# EPICS substitutions: iocCollimatorControl/R15CLM.substitutions
#R15CLM_BO,EPICS->PLC,Command
file "../../db/bo_word.template"{ pattern
{	P,		R,					PORT,		OFFSET,		MASK,		ZNAM,		ONAM	}
{	SR:R15:CLM:R15CLM:,	btn_LocalOrRemote,			R15CLM_BO1_Bits,	0,		0x0001,		Low,		High	}
{	SR:R15:CLM:R15CLM:,	btn_E_STOP,				R15CLM_BO1_Bits,	0,		0x0002,		Low,		High	}
{	SR:R15:CLM:R15CLM:,	m_restartTC,				R15CLM_BO1_Bits,	0,		0x0004,		Low,		High	}
{	SR:R15:CLM:R15CLM:,	btn_Move_Axis1,				R15CLM_BO2_Bits,	0,		0x0001,		Low,		High	}
{	SR:R15:CLM:R15CLM:,	btn_JogForward_Axis1,			R15CLM_BO2_Bits,	0,		0x0002,		Low,		High	}
{	SR:R15:CLM:R15CLM:,	btn_JogBackward_Axis1,			R15CLM_BO2_Bits,	0,		0x0004,		Low,		High	}
{	SR:R15:CLM:R15CLM:,	btn_Stop_Axis1,				R15CLM_BO2_Bits,	0,		0x0008,		Low,		High	}
{	SR:R15:CLM:R15CLM:,	btn_Reset_Axis1,			R15CLM_BO2_Bits,	0,		0x0010,		Low,		High	}
{	SR:R15:CLM:R15CLM:,	btn_SetPosition_Axis1,			R15CLM_BO2_Bits,	0,		0x0020,		Low,		High	}
{	SR:R15:CLM:R15CLM:,	LVDT1_FunctionOn,			R15CLM_BO2_Bits,	0,		0x0040,		Low,		High	}
{	SR:R15:CLM:R15CLM:,	LVDT1_ManualReleaseAlarm,		R15CLM_BO2_Bits,	0,		0x0080,		Low,		High	}
{	SR:R15:CLM:R15CLM:,	btn_Move_Axis2,				R15CLM_BO3_Bits,	0,		0x0001,		Low,		High	}
{	SR:R15:CLM:R15CLM:,	btn_JogForward_Axis2,			R15CLM_BO3_Bits,	0,		0x0002,		Low,		High	}
{	SR:R15:CLM:R15CLM:,	btn_JogBackward_Axis2,			R15CLM_BO3_Bits,	0,		0x0004,		Low,		High	}
{	SR:R15:CLM:R15CLM:,	btn_Stop_Axis2,				R15CLM_BO3_Bits,	0,		0x0008,		Low,		High	}
{	SR:R15:CLM:R15CLM:,	btn_Reset_Axis2,			R15CLM_BO3_Bits,	0,		0x0010,		Low,		High	}
{	SR:R15:CLM:R15CLM:,	btn_SetPosition_Axis2,			R15CLM_BO3_Bits,	0,		0x0020,		Low,		High	}
{	SR:R15:CLM:R15CLM:,	LVDT2_FunctionOn,			R15CLM_BO3_Bits,	0,		0x0040,		Low,		High	}
{	SR:R15:CLM:R15CLM:,	LVDT2_ManualReleaseAlarm,		R15CLM_BO3_Bits,	0,		0x0080,		Low,		High	}
{	SR:R15:CLM:R15CLM:,	btn_Move_AxisAll,			R15CLM_BO4_Bits,	0,		0x0001,		Low,		High	}
{	SR:R15:CLM:R15CLM:,	btn_JogForward_AxisAll,			R15CLM_BO4_Bits,	0,		0x0002,		Low,		High	}
{	SR:R15:CLM:R15CLM:,	btn_JogBackward_AxisAll,		R15CLM_BO4_Bits,	0,		0x0004,		Low,		High	}
{	SR:R15:CLM:R15CLM:,	btn_Stop_AxisAll,			R15CLM_BO4_Bits,	0,		0x0008,		Low,		High	}
{	SR:R15:CLM:R15CLM:,	btn_Reset_AxisAll,			R15CLM_BO4_Bits,	0,		0x0010,		Low,		High	}
}
#R15CLM_AO,EPICS->PLC,Command
file "../../db/aoFloat64.template" { pattern
{	P,           	R,               			PORT,      	OFFSET,   	DATA_TYPE,    	LOPR, 	HOPR, PREC	}
{	SR:R15:CLM:R15CLM:,	targetPositionAxis1,			R15CLM_AO1_FLOAT,	0,		FLOAT32_LE,	-1e6,	1e6,	4	}
{	SR:R15:CLM:R15CLM:,	targetVelocityAxis1,			R15CLM_AO1_FLOAT,	2,		FLOAT32_LE,	-1e6,	1e6,	4	}
{	SR:R15:CLM:R15CLM:,	increaseJogPositionAxis1,		R15CLM_AO1_FLOAT,	4,		FLOAT32_LE,	-1e6,	1e6,	4	}
{	SR:R15:CLM:R15CLM:,	Axis1_minPosition,			R15CLM_AO1_FLOAT,	6,		FLOAT32_LE,	-1e6,	1e6,	4	}
{	SR:R15:CLM:R15CLM:,	Axis1_maxPosition,			R15CLM_AO1_FLOAT,	8,		FLOAT32_LE,	-1e6,	1e6,	4	}
{	SR:R15:CLM:R15CLM:,	LVDT1_Threshold,			R15CLM_AO1_FLOAT,	10,		FLOAT32_LE,	-1e6,	1e6,	4	}
{	SR:R15:CLM:R15CLM:,	PositionSetValue_Axis1,			R15CLM_AO1_FLOAT,	12,		FLOAT32_LE,	-1e6,	1e6,	4	}
{	SR:R15:CLM:R15CLM:,	targetPositionAxis2,			R15CLM_AO2_FLOAT,	0,		FLOAT32_LE,	-1e6,	1e6,	4	}
{	SR:R15:CLM:R15CLM:,	targetVelocityAxis2,			R15CLM_AO2_FLOAT,	2,		FLOAT32_LE,	-1e6,	1e6,	4	}
{	SR:R15:CLM:R15CLM:,	increaseJogPositionAxis2,		R15CLM_AO2_FLOAT,	4,		FLOAT32_LE,	-1e6,	1e6,	4	}
{	SR:R15:CLM:R15CLM:,	Axis2_minPosition,			R15CLM_AO2_FLOAT,	6,		FLOAT32_LE,	-1e6,	1e6,	4	}
{	SR:R15:CLM:R15CLM:,	Axis2_maxPosition,			R15CLM_AO2_FLOAT,	8,		FLOAT32_LE,	-1e6,	1e6,	4	}
{	SR:R15:CLM:R15CLM:,	LVDT2_Threshold,			R15CLM_AO2_FLOAT,	10,		FLOAT32_LE,	-1e6,	1e6,	4	}
{	SR:R15:CLM:R15CLM:,	PositionSetValue_Axis2,			R15CLM_AO2_FLOAT,	12,		FLOAT32_LE,	-1e6,	1e6,	4	}
}
#R15CLM_BI,PLC->EPICS,Respond
file "../../db/bi_word.template"{ pattern
{	P,		R,					PORT,		OFFSET,		MASK,		ZNAM,		ONAM,		ZSV,		OSV,		SCAN		}
{	SR:R15:CLM:R15CLM:,	E_STOP_led,				R15CLM_BI1_Bits,	0,		0x0001,		Low,		High,		NO_ALARM,	NO_ALARM,	"I/O Intr"	}
{	SR:R15:CLM:R15CLM:,	Local_led,				R15CLM_BI1_Bits,	0,		0x0002,		Low,		High,		NO_ALARM,	NO_ALARM,	"I/O Intr"	}
{	SR:R15:CLM:R15CLM:,	Remote_led,				R15CLM_BI1_Bits,	0,		0x0004,		Low,		High,		NO_ALARM,	NO_ALARM,	"I/O Intr"	}
{	SR:R15:CLM:R15CLM:,	Error_led,				R15CLM_BI1_Bits,	0,		0x0008,		Low,		High,		NO_ALARM,	NO_ALARM,	"I/O Intr"	}
{	SR:R15:CLM:R15CLM:,	Axis1_error,				R15CLM_BI2_Bits,	0,		0x0001,		Low,		High,		NO_ALARM,	NO_ALARM,	"I/O Intr"	}
{	SR:R15:CLM:R15CLM:,	Axis1_moving,				R15CLM_BI2_Bits,	0,		0x0002,		Low,		High,		NO_ALARM,	NO_ALARM,	"I/O Intr"	}
{	SR:R15:CLM:R15CLM:,	foreward_limit_axis1,			R15CLM_BI2_Bits,	0,		0x0004,		Low,		High,		NO_ALARM,	NO_ALARM,	"I/O Intr"	}
{	SR:R15:CLM:R15CLM:,	backward_limit_axis1,			R15CLM_BI2_Bits,	0,		0x0008,		Low,		High,		NO_ALARM,	NO_ALARM,	"I/O Intr"	}
{	SR:R15:CLM:R15CLM:,	Moving_done_Axis1,			R15CLM_BI2_Bits,	0,		0x0010,		Low,		High,		NO_ALARM,	NO_ALARM,	"I/O Intr"	}
{	SR:R15:CLM:R15CLM:,	PositionSetDone_Axis1,			R15CLM_BI2_Bits,	0,		0x0020,		Low,		High,		NO_ALARM,	NO_ALARM,	"I/O Intr"	}
{	SR:R15:CLM:R15CLM:,	Axis2_error,				R15CLM_BI3_Bits,	0,		0x0001,		Low,		High,		NO_ALARM,	NO_ALARM,	"I/O Intr"	}
{	SR:R15:CLM:R15CLM:,	Axis2_moving,				R15CLM_BI3_Bits,	0,		0x0002,		Low,		High,		NO_ALARM,	NO_ALARM,	"I/O Intr"	}
{	SR:R15:CLM:R15CLM:,	foreward_limit_axis2,			R15CLM_BI3_Bits,	0,		0x0004,		Low,		High,		NO_ALARM,	NO_ALARM,	"I/O Intr"	}
{	SR:R15:CLM:R15CLM:,	backward_limit_axis2,			R15CLM_BI3_Bits,	0,		0x0008,		Low,		High,		NO_ALARM,	NO_ALARM,	"I/O Intr"	}
{	SR:R15:CLM:R15CLM:,	Moving_done_Axis2,			R15CLM_BI3_Bits,	0,		0x0010,		Low,		High,		NO_ALARM,	NO_ALARM,	"I/O Intr"	}
{	SR:R15:CLM:R15CLM:,	PositionSetDone_Axis2,			R15CLM_BI3_Bits,	0,		0x0020,		Low,		High,		NO_ALARM,	NO_ALARM,	"I/O Intr"	}
}
#R15CLM_AI,PLC->EPICS,Respond
file "../../db/aiFloat64.template"{ pattern
{	P,			R,					PORT,		OFFSET,		DATA_TYPE,	LOPR,	HOPR,	PREC,	SCAN			}
{	SR:R15:CLM:R15CLM:,	Axis1_Currentvelocity,			R15CLM_AI1_FLOAT,	0,		FLOAT32_LE,	-1e6,	1e6,	4,	"I/O Intr"		}
{	SR:R15:CLM:R15CLM:,	Axis1_CurrentPosition,			R15CLM_AI1_FLOAT,	2,		FLOAT32_LE,	-1e6,	1e6,	4,	"I/O Intr"		}
{	SR:R15:CLM:R15CLM:,	LVDT1_PV,				R15CLM_AI1_FLOAT,	4,		FLOAT32_LE,	-1e6,	1e6,	4,	"I/O Intr"		}
{	SR:R15:CLM:R15CLM:,	Axis2_Currentvelocity,			R15CLM_AI2_FLOAT,	0,		FLOAT32_LE,	-1e6,	1e6,	4,	"I/O Intr"		}
{	SR:R15:CLM:R15CLM:,	Axis2_CurrentPosition,			R15CLM_AI2_FLOAT,	2,		FLOAT32_LE,	-1e6,	1e6,	4,	"I/O Intr"		}
{	SR:R15:CLM:R15CLM:,	LVDT2_PV,				R15CLM_AI2_FLOAT,	4,		FLOAT32_LE,	-1e6,	1e6,	4,	"I/O Intr"		}
}
#R15CLM_Intin,PLC->EPICS,Respond
file "../../db/int64in.template"{ pattern
{	P,			R,			PORT,		OFFSET,		DATA_TYPE,	SCAN			}
{	SR:R15:CLM:R15CLM:,	ErrorId,		R15CLM_Intin,		0,		INT32_LE,	"I/O Intr"		}
}
#StringIn,PLC->EPICS,Respond
file "../../db/stringin.template"{ pattern
{	P,			R,				PORT,		OFFSET,		DATA_TYPE,	SCAN			}
{	SR:R15:CLM:R15CLM:,	ErrorDescription,		R15CLM_Stringin,	0,		STRING_LOW_HIGH,		"I/O Intr"		}
}
